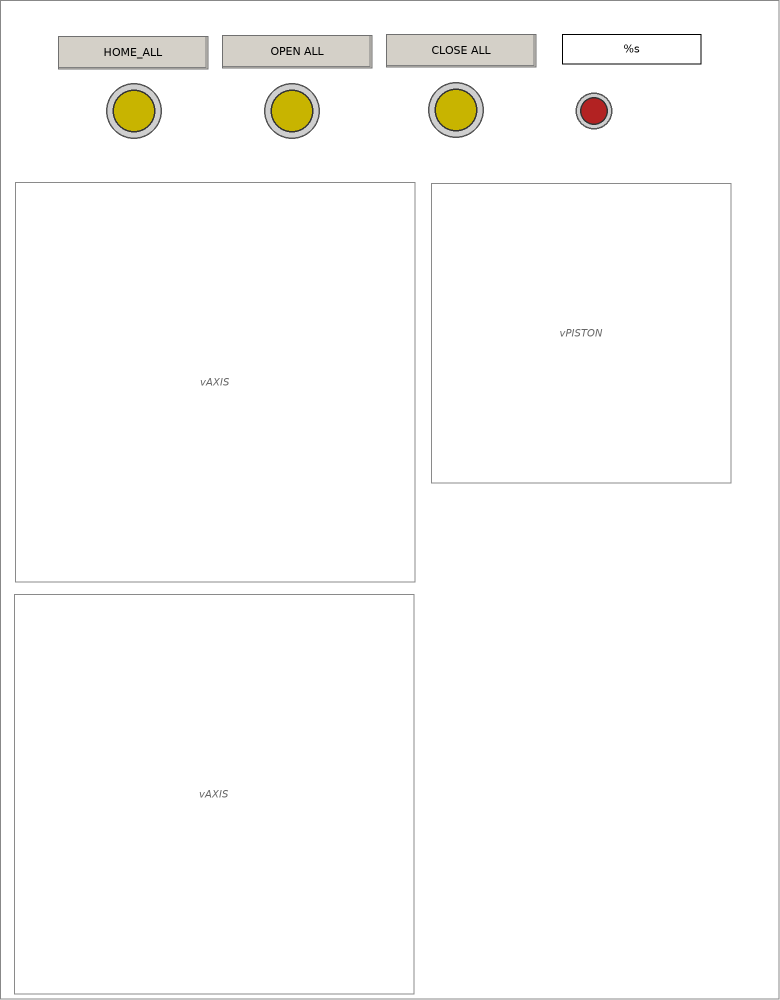
VISUALIZATION vACTION  // 780x1000
VAR_IN_OUT
	vACTION:FB_ACTION;
END_VAR
    Frame (15,182 400x400)
        shows vAXIS(vAxis := vACTION.aLIFT)
    Frame (431,183 300x300)
        shows vPISTON(PIST1 := vACTION.PIST)
    Frame (14,594 400x400)
        shows vAXIS(vAxis := vACTION.aXY)
    Button (58,36 150x33), "HOME_ALL"
        OnMouseDown: execute { vACTION.bHOME_ALL:=TRUE; }
    Lamp1 (102,79 64x64), variable: vACTION.bALL_HOMED, style: Lamp-Lamp1-Yellow
    Button (222,35 150x33), "OPEN ALL"
        OnMouseDown: execute { vACTION.bOPEN_ALL:=TRUE; }
    Lamp1 (260,79 64x64), variable: vACTION.bALL_OPENED, style: Lamp-Lamp1-Yellow
    Button (386,34 150x33), "CLOSE ALL"
        OnMouseDown: execute { vACTION.bCLOSE_ALL:=TRUE; }
    Lamp1 (424,78 64x64), variable: vACTION.bALL_CLOSED, style: Lamp-Lamp1-Yellow
    Lamp1 (573,88 42x46), variable: vACTION.bACTION_ERROR, style: Lamp-Lamp1-Red
    Rectangle (562,34 139x30), "%s", text variable: vACTION.sACTION_STATE
END_VISUALIZATION

(* stored: Version 1.1.0.1, ProductVersion 3.1.4024.12
   Visu vACTION: Id {d21375e2-c764-44f8-9c50-3c770c1388ac} *)
